// TIA Portal project "scl_kesikli_sürekli çalıştırma" (V18)

(* hardware
DEVICE "S7-1200 station_1"  S7-1200 Station
   slot 0: "Rack_0"  S7-1200 Rack  Rack  V1.0
   slot 1: "PLC_1"  CPU 1214C DC/DC/DC  6ES7 214-1AG40-0XB0  V4.6
*)

// ===== PLC "PLC_1"  CPU 1214C DC/DC/DC =====

VAR_GLOBAL   // PLC tag table "Default tag table"
   "KESİK BUTON" AT %I0.1 : Bool;
   "SÜREKLİ BUTON" AT %I0.2 : Bool;
   "STOP" AT %I0.3 : Bool;
   "MOTOR" AT %Q0.0 : Bool;
   "YARDIMCI RÖLE" AT %M0.0 : Bool;
END_VAR

FUNCTION "Block_1" : Void   // FC1, SCL
{ S7_Optimized_Access := 'TRUE' }
VERSION : 0.1
BEGIN
   IF "KESİK BUTON"=1 OR "YARDIMCI RÖLE"=1  THEN
       "MOTOR" := 1;
   ELSE
       "MOTOR" := 0;
   END_IF;

   IF "SÜREKLİ BUTON"=1 THEN
       "YARDIMCI RÖLE" := 1;

   END_IF;

   IF "STOP"=1 THEN
       "YARDIMCI RÖLE" := 0;
   ELSE
       // Statement section ELSE
       ;
   END_IF;
END_FUNCTION

ORGANIZATION_BLOCK "Main"   // OB1, LAD, ProgramCycle
TITLE = "Main Program Sweep (Cycle)"
{ S7_Optimized_Access := 'TRUE' }
VERSION : 0.1
// UGULAMA-2: Kesik-Sürekli Çalistirma.
// •*I0.1 butonu ile Q0.0 qikisi kesik çalisir.
// -*I0.2 butonu ile Q0.0 gikisi sürekli çalisir.
// -*I0.3 butonu ile Q0.0 cikisi durur.
   VAR_INPUT
      Initial_Call : Bool;   // Initial call of this OB
      Remanence : Bool;   // =True, if remanent data are available
   END_VAR
BEGIN

REGION Network 1
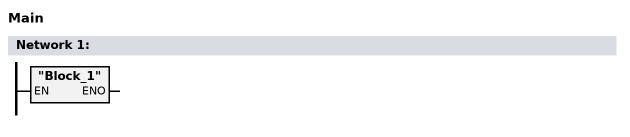
   RUNG wire#powerrail
      "Block_1"()
   END_RUNG
   // the same network as SCL:
   "Block_1"();
END_REGION
END_ORGANIZATION_BLOCK